# EPICS StreamDevice protocol: iocs/estherVacuum/vacApp/Db/inficonVG401.proto
Terminator = CR LF;
ReplyTimeout = 2000;
MaxInput     = 100;

#0, 1.0000E+03 mbar

EnablePressure {
   out "COM,1";
   in ACK;
}

ReadPressure {
    in "%(\$1)u, %E mBar";
}
